// TIA Portal V19 export
ORGANIZATION_BLOCK "TOD_INT0"   // OB10, LAD, TimeOfDay
TITLE = "Time of Day Interrupt"
   VAR_TEMP
      OB10_EV_CLASS : Byte;   // Bits 0-3 = 1 (Coming event), Bits 4-7 = 1 (Event class 1)
      OB10_STRT_INFO : Byte;   // 16#11 (OB 10 has started)
      OB10_PRIORITY : Byte;   // Priority of OB Execution
      OB10_OB_NUMBR : Byte;   // 10 (Organization block 10, OB10)
      OB10_RESERVED_1 : Byte;   // Reserved for system
      OB10_RESERVED_2 : Byte;   // Reserved for system
      OB10_PERIOD_EXE : Word;   // Period of execution (once, per minute/hour/day/week/month/year)
      OB10_RESERVED_3 : Int;   // Reserved for system
      OB10_RESERVED_4 : Int;   // Reserved for system
      OB10_DATE_TIME : Date_And_Time;   // Date and time OB10 started
   END_VAR
BEGIN

REGION Network 1
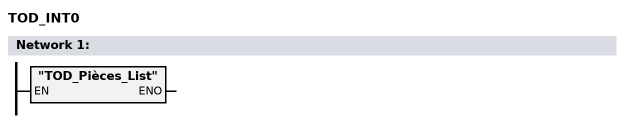
   RUNG wire#powerrail
      "TOD_Pièces_List"()
   END_RUNG
   // the same network as SCL:
   "TOD_Pièces_List"();
END_REGION
END_ORGANIZATION_BLOCK
